PROGRAM DataAcquisition
VAR
END_VAR


RunMATLAB();
ReadWriteOPCvariables();

END_PROGRAM

(* stored: Version 1.1.0.1, ProductVersion 3.1.4024.9
   POU DataAcquisition: Id {8ef7b23d-377f-464a-94da-dbf13a683f44}, SpecialFunc None *)
